FUNCTION F_AlarmLog : BOOL
VAR_INPUT
	iLevel: INT;
	sName : STRING;
	bNew  : BOOL;
END_VAR
VAR
	
END_VAR
VAR_IN_OUT
	bOld : BOOL;
END_VAR

IF (bOld <> bNew) THEN
	Logging.fbAlarmLog.P_sModule := 'Alarm Toggled';
	Logging.fbAlarmLog.M_nLogger(iLogLevel:= Logging.fbAlarmLog.P_iLogVerbosity, 
								sSource:= sName , sMessage:=  F_Concat3(BOOL_TO_STRING(bOld),'->',BOOL_TO_STRING(bNew)));
	bOld := bNew;
END_IF

END_FUNCTION

(* stored: Version 1.1.0.1, ProductVersion 3.1.4022.18
   POU F_AlarmLog: Id {88bb64c1-1847-4501-b557-8e61a4f87b6c}, SpecialFunc None *)
